FUNCTION_BLOCK DO_4 (* Identifier for the output module *)
  (* Standard: 61499-2 *)
  (* Version 0.0, 2014-01-12, 4DIAC-IDE, 4DIAC-Consortium *)
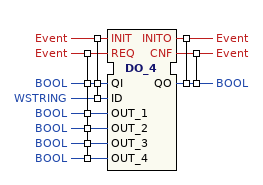
  EVENT_INPUT
    INIT WITH QI, ID; (* Initialization Request *)
    REQ WITH QI, OUT_1, OUT_2, OUT_3, OUT_4; (* Normal Execution Request *)
  END_EVENT
  EVENT_OUTPUT
    INITO WITH QO; (* Initialization Confirm *)
    CNF WITH QO; (* Execution Confirmation *)
  END_EVENT
  VAR_INPUT
    QI : BOOL; (* Input event qualifier *)
    ID : WSTRING; (* Identifier for the output module *)
    OUT_1 : BOOL;
    OUT_2 : BOOL;
    OUT_3 : BOOL;
    OUT_4 : BOOL;
  END_VAR
  VAR_OUTPUT
    QO : BOOL; (* Output event qualifier *)
  END_VAR
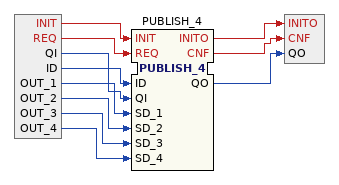
  FBS
    PUBLISH_4 : PUBLISH_4;
  END_FBS
  EVENT_CONNECTIONS
    INIT TO PUBLISH_4.INIT;
    REQ TO PUBLISH_4.REQ;
    PUBLISH_4.INITO TO INITO;
    PUBLISH_4.CNF TO CNF;
  END_CONNECTIONS
  DATA_CONNECTIONS
    ID TO PUBLISH_4.ID;
    QI TO PUBLISH_4.QI;
    OUT_1 TO PUBLISH_4.SD_1;
    OUT_2 TO PUBLISH_4.SD_2;
    OUT_3 TO PUBLISH_4.SD_3;
    OUT_4 TO PUBLISH_4.SD_4;
    PUBLISH_4.QO TO QO;
  END_CONNECTIONS
END_FUNCTION_BLOCK
